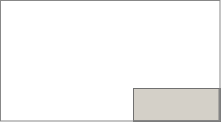
VISUALIZATION Visualization  // 221x122
    Button (133,88 88x34)
END_VISUALIZATION

(* stored: Version 1.1.0.1, ProductVersion 3.1.4024.6
   Visu Visualization: Id {2bf47564-407d-47e8-bd9e-f4d1432c7a7f} *)
